// TIA Portal V16 export
// export: Created 2021-07-12T14:47:20.6220706Z, ExportSetting WithDefaults, DisplayName Totally Integrated Automation Portal, DisplayVersion V16, DisplayName TIA Portal Version Control Interface, DisplayVersion V16, DisplayName TIA Portal Openness, DisplayVersion V16, DisplayName STEP 7 Professional, DisplayVersion V16, DisplayName STEP 7 Safety, DisplayVersion V16, DisplayName WinCC Professional, DisplayVersion V16
TYPE "SimaHydTO_typeHMIConnectionHmiDataVChar"
TITLE = SimaHydTO_typeHMIConnectionHmiDataVChar
// HMI interface: Calculated positions of VHar to display on HMI
// stored: IsFailsafeCompliant false
   STRUCT
      HMI_VChar : Array[1..200] of Real;
      HMI_VChar_MinQOutput : Real;
      HMI_VChar_MaxQOutput : Real;
      HMI_VChar_MinVelocity : Real;
      HMI_VCHar_MaxVelocity : Real;
      HMI_VChar_TrendRequest : Word;
      HMI_VChar_TrendTransfer : Word;
   END_STRUCT;
END_TYPE
